// TIA Portal V20 export
TYPE "UDT_Informe_DispositivoMaquina"
   STRUCT
      Prioridad : UInt;
      Bits : Struct
         Habilitado : Bool;
         DesHabilitado : Bool;
      END_STRUCT;
   END_STRUCT;
END_TYPE
